Omron CX-Programmer project NewProject (CX-Programmer 9.61)

# PLC NewPLC1: CP1L-E EM

## Global symbols (name address type ; comment)
0.00 BOOL  ; SEL MAN AUTO
0.02 BOOL  ; ALLARME INVERTER
0.03 BOOL  ; FUNGO
0.04 BOOL  ; EMERGENZA OK
1 CHANNEL  ; Register number
100.03 BOOL  ; CONSENSO A LINEA
253.13 BOOL  ; System Normally On Flag
30.01 BOOL  ; PUL TOUCHLAYOUT DX SX
30.02 BOOL  ; PUL PARAMETRI TOUCH
31.02 BOOL  ; Difd Output Pezzo
31.03 BOOL  ; MEM GO INV INGRESSO
31.04 BOOL  ; MEM GO INV CENTRALE
31.05 BOOL  ; MEM GO INV USCITA
31.06 BOOL  ; MEM STANDBY
31.07 BOOL  ; SCARICO VELOCE
31.10 BOOL  ; FINE SCANDEGGIO
31.11 BOOL  ; UP 0.02
31.12 BOOL  ; DOWN 0.02
31.13 BOOL  ; P_0_01s
41 CHANNEL  ; CANALE MANUALI
41.00 BOOL  ; MAN INGRESSO
41.01 BOOL  ; MAN CENTRALE
41.02 BOOL  ; MAN USCITA
50 CHANNEL  ; CanaleAllarme
50.01 BOOL  ; ConsensoValle
50.02 BOOL  ; Fungo Premuti
50.03 BOOL  ; Emergenza da esterno saltata
50.04 BOOL  ; AllarmeInverter
50.05 BOOL  ; TimeOutFoto312
50.06 BOOL  ; TimeOutFoto313
50.07 BOOL  ; TimeOutFoto314
50.08 BOOL  ; All.Temp.Minima
50.09 BOOL  ; All.Temp.Massima
A531.00 BOOL  ; reset counter
A640.00 BOOL  ; StartCom
A640.01 BOOL  ; ComOk
A640.02 BOOL  ; ComError
C0051 BOOL  ; DURATA TEMPO SCANDEGGIO VELOCE
C0052 BOOL  ; Rit.ConsensoDaLinea
D32300 CHANNEL  ; slave number
D32301 CHANNEL  ; function code
D32302 CHANNEL  ; data bytes
D32303 CHANNEL  ; register number
D32304 CHANNEL  ; number of registers to be writin
D32305 CHANNEL  ; attatched data size in bytes
D32306 CHANNEL  ; Operation command
D32307 CHANNEL  ; Frequancy
W0.00 BOOL  ; start1
W0.01 BOOL  ; start2
W0.02 BOOL  ; start3
W0.03 BOOL  ; STOP
W10.00 BOOL  ; slave1 write
_0MINUS02_SEC_PULSE 254.01 BOOL  ; System 0.02 second clock pulse bit

## Program NewProgram1 (cyclic task 0)
Local symbols
P_Gt BOOL

### Section main

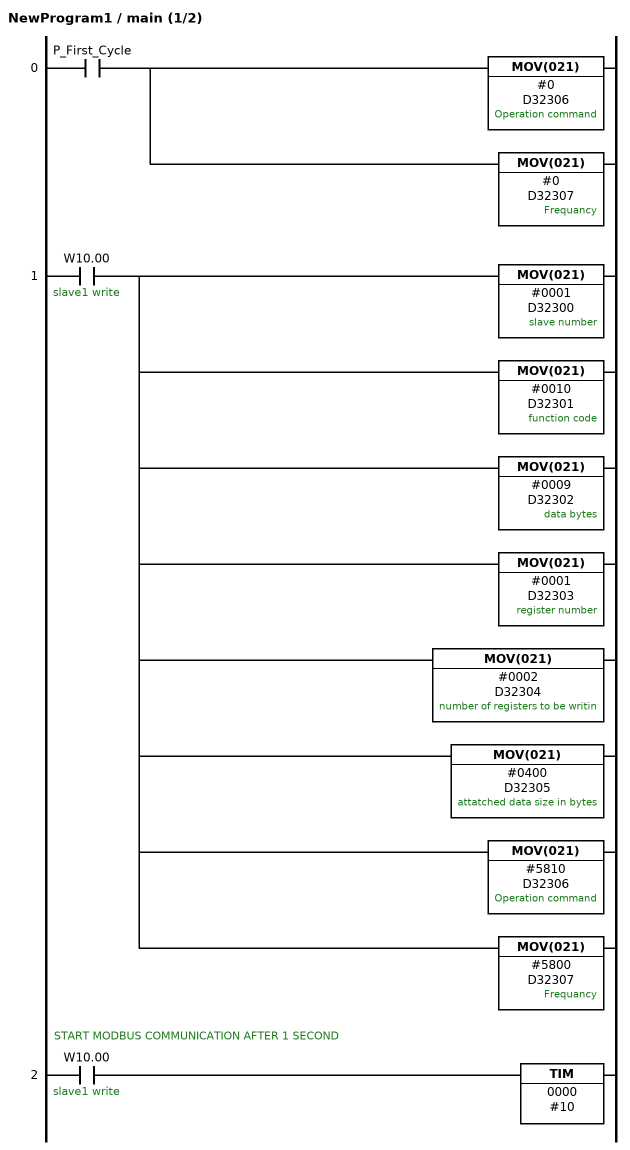
; rung 0
LD P_First_Cycle
MOV(021) #0 D32306  ; Operation command  // stop command (0)=Stop
MOV(021) #0 D32307  ; Frequancy  // Frequancy =0
; rung 1
LD W10.00  ; slave1 write
MOV(021) #0001 D32300  ; slave number
MOV(021) #0010 D32301  ; function code
MOV(021) #0009 D32302  ; data bytes
MOV(021) #0001 D32303  ; register number
MOV(021) #0002 D32304  ; number of registers to be writin
MOV(021) #0400 D32305  ; attatched data size in bytes
MOV(021) #5810 D32306  ; Operation command
MOV(021) #5800 D32307  ; Frequancy
; rung 2: START MODBUS COMMUNICATION AFTER 1 SECOND
LD W10.00  ; slave1 write
TIM 0000 #10

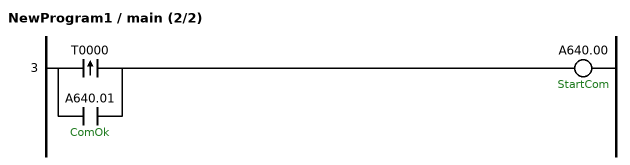
; rung 3
@LD T0000
OR A640.01  ; ComOk  // Modbus -RTU easy master function execution Normal flag
OUT A640.00  ; StartCom  // Modbus -RTU easy master function execution bit
; rung 4
END(001)